ABB RAPID module: Module1.mod

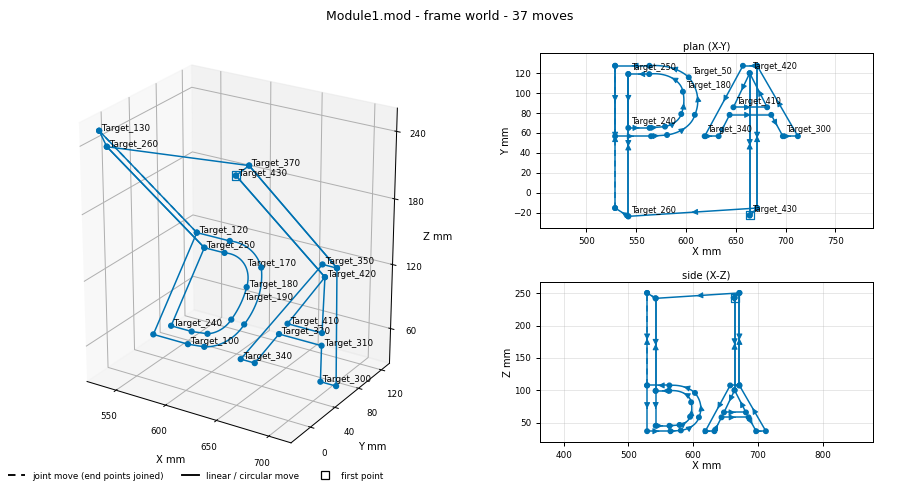
[picture p0: tool path of Module1.mod in frame world, 37 of 39 moves have a stored position in this frame; points joined in program order, loops and branches not executed]
MODULE Module1
        CONST robtarget Target_430:=[[-163.904,56.491,200],[0.160429997,-0.909843727,0.37686961,-0.06645228],[0,0,0,0],[9E+09,9E+09,9E+09,9E+09,9E+09,9E+09]];
    CONST robtarget Target_420:=[[-163.904,56.491,-2],[0.160429997,-0.909843727,0.37686961,-0.06645228],[0,0,0,0],[9E+09,9E+09,9E+09,9E+09,9E+09,9E+09]];
    CONST robtarget Target_410:=[[-147.533,104.922,-2],[0.160429997,-0.909843727,0.37686961,-0.06645228],[0,0,0,0],[9E+09,9E+09,9E+09,9E+09,9E+09,9E+09]];
    CONST robtarget Target_400:=[[-181.435,104.922,-2],[0.160429997,-0.909843727,0.37686961,-0.06645228],[0,0,0,0],[9E+09,9E+09,9E+09,9E+09,9E+09,9E+09]];
    CONST robtarget Target_390:=[[-163.904,56.491,-2],[0.160429997,-0.909843727,0.37686961,-0.06645228],[0,0,0,0],[9E+09,9E+09,9E+09,9E+09,9E+09,9E+09]];
    CONST robtarget Target_380:=[[-163.904,56.491,200],[0.160429997,-0.909843727,0.37686961,-0.06645228],[0,0,0,0],[9E+09,9E+09,9E+09,9E+09,9E+09,9E+09]];
    CONST robtarget Target_370:=[[-171.339,45.986,200],[0.160429997,-0.909843727,0.37686961,-0.06645228],[0,0,0,0],[9E+09,9E+09,9E+09,9E+09,9E+09,9E+09]];
    CONST robtarget Target_360:=[[-171.339,45.986,-2],[0.160429997,-0.909843727,0.37686961,-0.06645228],[0,0,0,0],[9E+09,9E+09,9E+09,9E+09,9E+09,9E+09]];
    CONST robtarget Target_350:=[[-157.083,45.986,-2],[0.160429997,-0.909843727,0.37686961,-0.06645228],[0,0,0,0],[9E+09,9E+09,9E+09,9E+09,9E+09,9E+09]];
    CONST robtarget Target_340:=[[-118.679,145.986,-2],[0.160429997,-0.909843727,0.37686961,-0.06645228],[0,0,0,0],[9E+09,9E+09,9E+09,9E+09,9E+09,9E+09]];
    CONST robtarget Target_330:=[[-132.731,145.986,-2],[0.160429997,-0.909843727,0.37686961,-0.06645228],[0,0,0,0],[9E+09,9E+09,9E+09,9E+09,9E+09,9E+09]];
    CONST robtarget Target_320:=[[-143.713,115.7,-2],[0.160429997,-0.909843727,0.37686961,-0.06645228],[0,0,0,0],[9E+09,9E+09,9E+09,9E+09,9E+09,9E+09]];
    CONST robtarget Target_310:=[[-185.527,115.7,-2],[0.160429997,-0.909843727,0.37686961,-0.06645228],[0,0,0,0],[9E+09,9E+09,9E+09,9E+09,9E+09,9E+09]];
    CONST robtarget Target_300:=[[-197.192,145.986,-2],[0.160429997,-0.909843727,0.37686961,-0.06645228],[0,0,0,0],[9E+09,9E+09,9E+09,9E+09,9E+09,9E+09]];
    CONST robtarget Target_290:=[[-212.267,145.986,-2],[0.160429997,-0.909843727,0.37686961,-0.06645228],[0,0,0,0],[9E+09,9E+09,9E+09,9E+09,9E+09,9E+09]];
    CONST robtarget Target_280:=[[-171.339,45.986,-2],[0.160429997,-0.909843727,0.37686961,-0.06645228],[0,0,0,0],[9E+09,9E+09,9E+09,9E+09,9E+09,9E+09]];
    CONST robtarget Target_270:=[[-171.339,45.986,200],[0.160429997,-0.909843727,0.37686961,-0.06645228],[0,0,0,0],[9E+09,9E+09,9E+09,9E+09,9E+09,9E+09]];
    CONST robtarget Target_260:=[[-42.008,57.787,200],[0.160429997,-0.909843727,0.37686961,-0.06645228],[0,0,0,0],[9E+09,9E+09,9E+09,9E+09,9E+09,9E+09]];
    CONST robtarget Target_250:=[[-42.008,57.787,-2],[0.160429997,-0.909843727,0.37686961,-0.06645228],[0,0,0,0],[9E+09,9E+09,9E+09,9E+09,9E+09,9E+09]];
    CONST robtarget Target_240:=[[-42.008,134.186,-2],[0.160429997,-0.909843727,0.37686961,-0.06645228],[0,0,0,0],[9E+09,9E+09,9E+09,9E+09,9E+09,9E+09]];
    CONST robtarget Target_230:=[[-63.358,134.186,-2],[0.160429997,-0.909843727,0.37686961,-0.06645228],[0,0,0,0],[9E+09,9E+09,9E+09,9E+09,9E+09,9E+09]];
    CONST robtarget Target_220:=[[-78.877,132.344,-2],[0.160429997,-0.909843727,0.37686961,-0.06645228],[0,0,0,0],[9E+09,9E+09,9E+09,9E+09,9E+09,9E+09]];
    CONST robtarget Target_210:=[[-87.847,127.16,-2],[0.160429997,-0.909843727,0.37686961,-0.06645228],[0,0,0,0],[9E+09,9E+09,9E+09,9E+09,9E+09,9E+09]];
    CONST robtarget Target_200:=[[-95.18,114.506,-2],[0.160429997,-0.909843727,0.37686961,-0.06645228],[0,0,0,0],[9E+09,9E+09,9E+09,9E+09,9E+09,9E+09]];
    CONST robtarget Target_190:=[[-97.806,95.236,-2],[0.160429997,-0.909843727,0.37686961,-0.06645228],[0,0,0,0],[9E+09,9E+09,9E+09,9E+09,9E+09,9E+09]];
    CONST robtarget Target_180:=[[-96.84,82.808,-2],[0.160429997,-0.909843727,0.37686961,-0.06645228],[0,0,0,0],[9E+09,9E+09,9E+09,9E+09,9E+09,9E+09]];
    CONST robtarget Target_170:=[[-87.328,64.425,-2],[0.160429997,-0.909843727,0.37686961,-0.06645228],[0,0,0,0],[9E+09,9E+09,9E+09,9E+09,9E+09,9E+09]];
    CONST robtarget Target_160:=[[-63.017,57.787,-2],[0.160429997,-0.909843727,0.37686961,-0.06645228],[0,0,0,0],[9E+09,9E+09,9E+09,9E+09,9E+09,9E+09]];
    CONST robtarget Target_150:=[[-42.008,57.787,-2],[0.160429997,-0.909843727,0.37686961,-0.06645228],[0,0,0,0],[9E+09,9E+09,9E+09,9E+09,9E+09,9E+09]];
    CONST robtarget Target_140:=[[-42.008,57.787,200],[0.160429997,-0.909843727,0.37686961,-0.06645228],[0,0,0,0],[9E+09,9E+09,9E+09,9E+09,9E+09,9E+09]];
    CONST robtarget Target_130:=[[-28.774,45.986,200],[0.160429997,-0.909843727,0.37686961,-0.06645228],[0,0,0,0],[9E+09,9E+09,9E+09,9E+09,9E+09,9E+09]];
    CONST robtarget Target_120:=[[-28.774,45.986,-2],[0.160429997,-0.909843727,0.37686961,-0.06645228],[0,0,0,0],[9E+09,9E+09,9E+09,9E+09,9E+09,9E+09]];
    CONST robtarget Target_110:=[[-28.774,145.986,-2],[0.160429997,-0.909843727,0.37686961,-0.06645228],[0,0,0,0],[9E+09,9E+09,9E+09,9E+09,9E+09,9E+09]];
    CONST robtarget Target_100:=[[-64.859,145.986,-2],[0.160429997,-0.909843727,0.37686961,-0.06645228],[0,0,0,0],[9E+09,9E+09,9E+09,9E+09,9E+09,9E+09]];
    CONST robtarget Target_90:=[[-80.923,144.281,-2],[0.160429997,-0.909843727,0.37686961,-0.06645228],[0,0,0,0],[9E+09,9E+09,9E+09,9E+09,9E+09,9E+09]];
    CONST robtarget Target_80:=[[-92.86,139.268,-2],[0.160429997,-0.909843727,0.37686961,-0.06645228],[0,0,0,0],[9E+09,9E+09,9E+09,9E+09,9E+09,9E+09]];
    CONST robtarget Target_70:=[[-108.788,115.632,-2],[0.160429997,-0.909843727,0.37686961,-0.06645228],[0,0,0,0],[9E+09,9E+09,9E+09,9E+09,9E+09,9E+09]];
    CONST robtarget Target_60:=[[-110.561,83.373,-2],[0.160429997,-0.909843727,0.37686961,-0.06645228],[0,0,0,0],[9E+09,9E+09,9E+09,9E+09,9E+09,9E+09]];
    CONST robtarget Target_50:=[[-102.716,62.354,-2],[0.160429997,-0.909843727,0.37686961,-0.06645228],[0,0,0,0],[9E+09,9E+09,9E+09,9E+09,9E+09,9E+09]];
    CONST robtarget Target_40:=[[-81.025,47.419,-2],[0.160429997,-0.909843727,0.37686961,-0.06645228],[0,0,0,0],[9E+09,9E+09,9E+09,9E+09,9E+09,9E+09]];
    CONST robtarget Target_30:=[[-63.222,45.986,-2],[0.160429997,-0.909843727,0.37686961,-0.06645228],[0,0,0,0],[9E+09,9E+09,9E+09,9E+09,9E+09,9E+09]];
    CONST robtarget Target_20:=[[-28.774,45.986,-2],[0.160429997,-0.909843727,0.37686961,-0.06645228],[0,0,0,0],[9E+09,9E+09,9E+09,9E+09,9E+09,9E+09]];
    CONST robtarget Target_10:=[[-28.774,45.986,200],[0.160429997,-0.909843727,0.37686961,-0.06645228],[0,0,0,0],[9E+09,9E+09,9E+09,9E+09,9E+09,9E+09]];
    CONST jointtarget JointTarget_1:=[[0,0,0,0,0,0],[9E+09,9E+09,9E+09,9E+09,9E+09,9E+09]];
!***********************************************************
    !
    ! Módulo:  Module1
    !
    ! Descripción:
    !   <Introduzca la descripción aquí>
    !
    ! Autor: sergi
    !
    ! Versión: 1.0
    !
    !***********************************************************


    !***********************************************************
    !
    ! Procedimiento Main
    !
    !   Este es el punto de entrada de su programa
    !
    !***********************************************************
    PROC main()
        !Añada aquí su código
        MoveAbsJ JointTarget_1,v1000,z100,lab1TCP\WObj:=Workobject_1;
        Path_lab1_SERDAN;
        MoveAbsJ JointTarget_1,v1000,z100,lab1TCP\WObj:=Workobject_1;
    ENDPROC
    PROC Path_lab1_SERDAN()
        MoveJ Target_430,v100,z10,lab1TCP\WObj:=Workobject_1;
        MoveL Target_420,v100,fine,lab1TCP\WObj:=Workobject_1;
        MoveL Target_410,v100,z10,lab1TCP\WObj:=Workobject_1;
        MoveL Target_400,v100,z10,lab1TCP\WObj:=Workobject_1;
        MoveL Target_390,v100,z10,lab1TCP\WObj:=Workobject_1;
        MoveL Target_380,v100,z10,lab1TCP\WObj:=Workobject_1;
        MoveL Target_370,v100,z10,lab1TCP\WObj:=Workobject_1;
        MoveL Target_360,v100,z10,lab1TCP\WObj:=Workobject_1;
        MoveL Target_350,v100,z10,lab1TCP\WObj:=Workobject_1;
        MoveL Target_340,v100,z10,lab1TCP\WObj:=Workobject_1;
        MoveL Target_330,v100,z10,lab1TCP\WObj:=Workobject_1;
        MoveL Target_320,v100,z10,lab1TCP\WObj:=Workobject_1;
        MoveL Target_310,v100,z10,lab1TCP\WObj:=Workobject_1;
        MoveL Target_300,v100,z10,lab1TCP\WObj:=Workobject_1;
        MoveL Target_290,v100,z10,lab1TCP\WObj:=Workobject_1;
        MoveL Target_280,v100,z10,lab1TCP\WObj:=Workobject_1;
        MoveL Target_270,v100,z10,lab1TCP\WObj:=Workobject_1;
        MoveL Target_260,v100,z10,lab1TCP\WObj:=Workobject_1;
        MoveL Target_250,v100,z10,lab1TCP\WObj:=Workobject_1;
        MoveL Target_240,v100,z10,lab1TCP\WObj:=Workobject_1;
        MoveL Target_230,v100,z10,lab1TCP\WObj:=Workobject_1;
        MoveL Target_220,v100,z10,lab1TCP\WObj:=Workobject_1;
        MoveC Target_210,Target_200,v100,z10,lab1TCP\WObj:=Workobject_1;
        MoveC Target_190,Target_180,v100,z10,lab1TCP\WObj:=Workobject_1;
        MoveC Target_170,Target_160,v100,z10,lab1TCP\WObj:=Workobject_1;
        MoveL Target_150,v100,z10,lab1TCP\WObj:=Workobject_1;
        MoveL Target_140,v100,z10,lab1TCP\WObj:=Workobject_1;
        MoveL Target_130,v100,z10,lab1TCP\WObj:=Workobject_1;
        MoveL Target_120,v100,z10,lab1TCP\WObj:=Workobject_1;
        MoveL Target_110,v100,z10,lab1TCP\WObj:=Workobject_1;
        MoveL Target_100,v100,z10,lab1TCP\WObj:=Workobject_1;
        MoveL Target_90,v100,z10,lab1TCP\WObj:=Workobject_1;
        MoveC Target_80,Target_70,v100,z10,lab1TCP\WObj:=Workobject_1;
        MoveC Target_60,Target_50,v100,z10,lab1TCP\WObj:=Workobject_1;
        MoveC Target_40,Target_30,v100,z10,lab1TCP\WObj:=Workobject_1;
        MoveL Target_20,v100,z10,lab1TCP\WObj:=Workobject_1;
        MoveJ Target_10,v100,z10,lab1TCP\WObj:=Workobject_1;
    ENDPROC
ENDMODULE
